PROGRAM MAIN
VAR
	IntVAr : INT;
	StrVar : STRING;
	FloatVar : REAL;
	RetunBytesINT : UDINT;
	RetunBytesSTR : UDINT;
	RetunBytesF : UDINT;
	
	nVariable : INT := 20;
	pPointer : POINTER TO INT := ADR(nVariable);
	RetunBytesPtr : UDINT;
	
	Variable : INT := 20;
	rReference : REFERENCE TO INT REF= Variable;
	RetunBytesRef : UDINT;
	aArray : ARRAY [1..5] OF INT := [10, 20, 30, 40, 50];
	nINT : INT;
END_VAR

RetunBytesINT := SIZEOF(IntVAr);
RetunBytesSTR := SIZEOF(StrVar);
RetunBytesF := SIZEOF(FloatVar);

pPointer^ := 30;
RetunBytesPtr := SIZEOF(pPointer);

rReference := 30;
RetunBytesRef := SIZEOF(rReference);

aArray[1] := 42;
nINT := aArray[1] + aArray[4];

END_PROGRAM

(* stored: Version 1.1.0.1, ProductVersion 3.1.4024.12
   POU MAIN: Id {efc4c9e5-0dae-4725-b959-1d5f1b22e40d}, SpecialFunc None *)
